FUNCTION_BLOCK FB_Discharge
VAR_INPUT
END_VAR
VAR_OUTPUT
END_VAR
VAR
		send_message : PTC_Send_Message;
		fbTimer : TON;
END_VAR

//Self resetting timer for calling for the command (put at an arbitrary 1s)
fbTimer(IN := NOT fbTimer.Q, PT := T#1S);

IF fbTimer.Q THEN
    send_message(ID := E_PTC_TX_ID.MAIN_FSM, Command := E_PTC_TX_Command.HV_OFF, CAN_OUTPUts := GVL_PT.CAN_OUTPUTS, CAN_INPUTS := GVL_PT.CAN_INPUTS);
END_IF

END_FUNCTION_BLOCK

(* stored: Version 1.1.0.1
   POU FB_Discharge: Id {9b334204-e1f0-4f77-8568-487de87d10d1}, SpecialFunc None *)
